// Mitsubishi GX Works2 project: CJ, 비상 명령   PLC: Q03UDV

PROGRAM MAIN
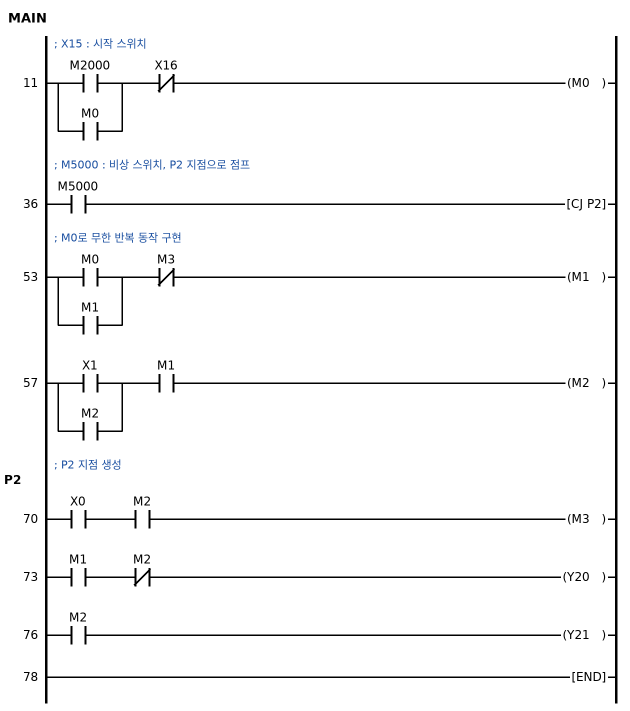
; X15 : 시작 스위치
11    LD      M2000
      OR      M0
      ANI     X16
      OUT     M0
; M5000 : 비상 스위치, P2 지점으로 점프
36    LD      M5000
      CJ      P2
; M0로 무한 반복 동작 구현
53    LD      M0
      OR      M1
      ANI     M3
      OUT     M1
57    LD      X1
      OR      M2
      AND     M1
      OUT     M2
      P2
; P2 지점 생성
70    LD      X0
      AND     M2
      OUT     M3
73    LD      M1
      ANI     M2
      OUT     Y20
76    LD      M2
      OUT     Y21
78    END
END_PROGRAM
